FUNCTION_BLOCK fbCalculateSetpoint
VAR_INPUT
	currentValue:REAL;
	nextSetpointValue:REAL;
	nextSetpointTime:LINT;
	currentSetpoint:REAL;
	previousSetpoint:REAL;
	previousSetpointTime:LINT;
	stepMode:BOOL;
	rampingMultiplier:REAL;
	bStepStart:BOOL;
END_VAR
VAR_OUTPUT
	setpoint:REAL;
	
END_VAR
VAR
	
	NextTemp: LREAL;
	
	nowMinutes: LINT;
	nowSeconds:LINT;
	now: TIMESTRUCT;
	fbTON: TON := (PT := TIME#1s0ms);
	
END_VAR


now := GVL.fbLocalSystemTime.systemTime;
nowMinutes := now.wHour*60+now.wMinute;
nowSeconds :=nowMinutes*60+now.wSecond;


fbTON();



IF stepMode=TRUE THEN
	
	IF nowMinutes >= nextSetpointTime THEN
		setpoint := nextSetpointValue;
	ELSE
		setpoint:=previousSetpoint;
	END_IF
	
ELSE

	//Ramp
	IF bStepStart THEN
	
		IF (nextSetpointTime-previousSetpointTime)<>0 THEN
			setpoint:= ((nextSetpointValue - previousSetpoint)/((nextSetpointTime-previousSetpointTime)))*(nowMinutes-previousSetpointTime)+previousSetpoint;
		END_IF
	
	ELSE
		IF ((nextSetpointTime*60)-nowSeconds)<>0 THEN
			setpoint:= ((nextSetpointValue - currentSetpoint)/(((nextSetpointTime*60)-nowSeconds)))*(GVL.cycleTime)+currentSetpoint;
		ELSIF ((nextSetpointTime*60)-nowSeconds)=0 THEN
			setpoint:=nextSetpointValue;
		END_IF
	END_IF
	
END_IF

END_FUNCTION_BLOCK

(* stored: Version 1.1.0.1, ProductVersion 3.1.4022.16
   POU fbCalculateSetpoint: Id {12b05b94-2f00-4d75-93a4-8438a88019e6}, SpecialFunc None *)
